// TIA Portal V19 export
DATA_BLOCK "RO 1 LEVEL DB"   // DB199
{ S7_Optimized_Access := 'FALSE' }
   VAR
      "AGLV 301 BUFF" : Int;
      "RECIRCULATION TIME SV" : Int;
      "RECIRCULATION TIME PV" : Int;
      "AGLV 302 BUFF" : Int;
      "RECIRCULATION TIME 302 SV" : Int;
      "RECIRCULATION TIME 302 PV" : Int;
      "LEVEL HI RECIRC BUFF" : Int;
      "LEVEL HI RECIRC RO ON TIME SV" : Int;
      "LEVEL HI RECIRC RO ON TIME PV" : Int;
      "LEVEL HI RECIRC RO OFF TIME SV" : Int;
      "LEVEL HI RECIRC RO OFF TIME PV" : Int;
   END_VAR
BEGIN
END_DATA_BLOCK
